Yaskawa INFORM job: B-8-08279-80-90-M.JBI

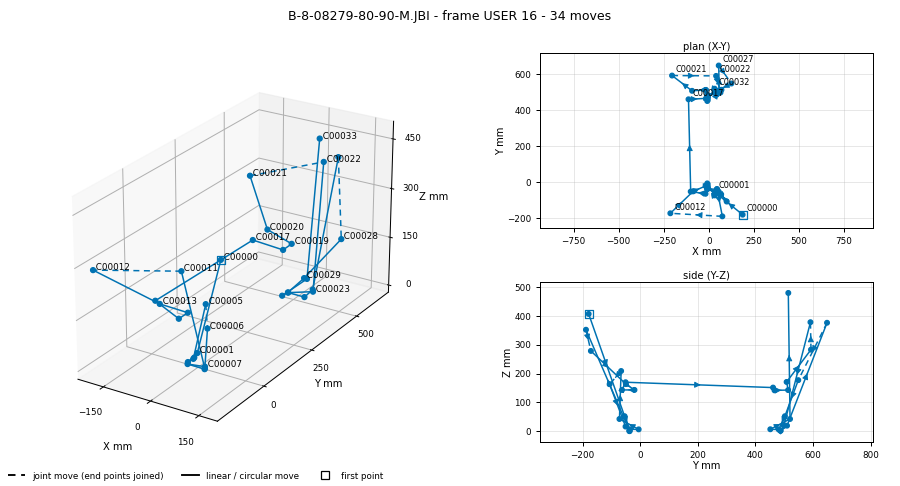
[picture p0: tool path of B-8-08279-80-90-M.JBI in frame USER 16, 34 of 34 moves have a stored position in this frame; points joined in program order, loops and branches not executed]
/JOB
//NAME B-8-08279-80-90-M
///FOLDERNAME PART_420-08279-80
//POS
///NPOS 34,0,34,0,0,0
///USER 16
///TOOL 4
///POSTYPE USER
///RECTAN
///RCONF 1,0,0,0,0,0,0,0,0,0,0,0,0,0,0,0,0,0,0,0,0,0,0,0
C00000=187.746,-179.018,407.228,-165.0003,45.0004,-0.0020
C00001=33.224,-54.308,52.156,-165.0000,45.0000,0.0000
C00002=-8.627,-36.453,6.455,-179.3917,57.1236,-36.5642
C00003=-8.579,-5.401,6.463,-179.4738,57.0912,-39.8725
C00004=32.283,-72.150,42.455,-165.0000,45.0000,0.0000
C00005=68.685,-66.272,209.042,-165.0000,45.0000,0.0000
C00006=99.538,-106.298,163.160,-166.3780,45.3490,-50.4350
C00007=54.868,-50.966,16.241,133.5610,7.6410,-152.0390
C00008=-9.081,-37.305,0.844,126.3818,11.5234,-151.1127
C00009=44.780,-37.124,0.073,126.4040,11.5044,-151.1169
C00010=45.512,-37.136,1.975,126.4030,11.5049,-151.1151
C00011=75.120,-188.373,352.355,175.5546,51.6267,-23.6686
C00012=-213.482,-171.326,278.744,154.4200,34.7310,45.4810
C00013=-87.212,-49.799,163.694,107.6090,9.3560,77.2190
C00014=-18.100,-19.955,143.362,104.0898,8.5656,76.6645
C00015=-18.153,-63.177,143.317,104.0907,8.5651,76.6651
C00016=-100.598,-50.810,170.079,107.6090,9.3560,77.2190
C00017=-112.794,461.129,151.518,107.5190,-7.4490,103.3910
C00018=-15.652,466.321,141.837,97.5692,-4.9506,104.4470
C00019=-15.525,513.463,142.905,97.5693,-4.9511,104.4481
C00020=-92.930,508.215,171.083,107.5190,-7.4490,103.3910
C00021=-203.967,592.873,283.205,107.5190,-7.4490,103.3910
C00022=40.454,590.981,378.479,-169.5230,46.0050,83.6620
C00023=64.926,498.805,18.936,-133.5620,7.6410,152.0390
C00024=-9.742,487.137,1.976,-127.4879,10.8527,151.2414
C00025=43.903,487.064,1.330,-127.4894,10.8533,151.2422
C00026=57.653,509.668,19.257,-133.5618,7.6414,152.0397
C00027=54.868,648.552,376.545,-169.5230,46.0050,83.6620
C00028=125.357,548.743,177.335,165.0000,45.0000,0.0000
C00029=33.224,502.241,52.156,165.0000,45.0000,0.0000
C00030=-7.002,480.856,5.907,165.0476,50.9832,6.6545
C00031=-8.581,451.633,6.779,162.6596,51.5731,19.7580
C00032=32.283,520.083,42.455,165.0000,45.0000,0.0000
C00033=70.181,514.089,480.075,165.0008,44.9999,-0.0009
///TOOL 0
///POSTYPE ANGLE
///ANGLE
EC00000=90.0000
///TOOL 4
EC00001=90.0000
///TOOL 0
EC00002=90.0000
EC00003=90.0000
///TOOL 4
EC00004=90.0000
EC00005=90.0000
EC00006=105.0000
EC00007=105.0000
///TOOL 0
EC00008=105.0000
EC00009=105.0000
EC00010=105.0000
EC00011=105.0000
///TOOL 4
EC00012=135.0000
EC00013=135.0000
///TOOL 0
EC00014=135.0000
EC00015=135.0000
///TOOL 4
EC00016=135.0000
EC00017=135.0000
///TOOL 0
EC00018=135.0000
EC00019=135.0000
///TOOL 4
EC00020=135.0000
EC00021=135.0000
EC00022=105.0000
EC00023=105.0000
///TOOL 0
EC00024=105.0000
EC00025=105.0000
EC00026=105.0000
///TOOL 4
EC00027=105.0000
EC00028=90.0000
EC00029=90.0000
///TOOL 0
EC00030=90.0000
EC00031=90.0000
///TOOL 4
EC00032=90.0000
///TOOL 0
EC00033=90.0000
//INST
///DATE 2021/10/29 11:36
///ATTR SC,RW,RJ
////FRAME USER 16
///GROUP1 RB1
///GROUP2 ST3
NOP
INC I005
'Path Start: PP1_1
MOVJ C00000 VJ=100.00  +MOVJ EC00000
SMOVL C00001 V=1250.0  +MOVJ EC00001
SMOVL C00002 V=1250.0  +MOVJ EC00002
ARCON ASF#(951)
SMOVL C00003 V=8.5  +MOVJ EC00003
ARCOF AEF#(951)
SMOVL C00004 V=1250.0  +MOVJ EC00004
SMOVL C00005 V=1250.0  +MOVJ EC00005
'Path End
'Path Start: PP48
MOVJ C00006 VJ=100.00  +MOVJ EC00006
SMOVL C00007 V=1250.0  +MOVJ EC00007
SMOVL C00008 V=300.0  +MOVJ EC00008
ARCON ASF#(953)
SMOVL C00009 V=15.7  +MOVJ EC00009
ARCOF AEF#(953)
SMOVL C00010 V=1250.0  +MOVJ EC00010
SMOVL C00011 V=1250.0  +MOVJ EC00011
'Path End
'Path Start: PP47
MOVJ C00012 VJ=100.00  +MOVJ EC00012
SMOVL C00013 V=1250.0  +MOVJ EC00013
SMOVL C00014 V=300.0  +MOVJ EC00014
ARCON ASF#(953)
SMOVL C00015 V=12.7  +MOVJ EC00015
ARCOF AEF#(953)
SMOVL C00016 V=1250.0  +MOVJ EC00016
'Path End
'Path Start: PP42
SMOVL C00017 V=1250.0  +MOVJ EC00017
SMOVL C00018 V=300.0  +MOVJ EC00018
ARCON ASF#(953)
SMOVL C00019 V=12.7  +MOVJ EC00019
ARCOF AEF#(953)
SMOVL C00020 V=1250.0  +MOVJ EC00020
SMOVL C00021 V=1250.0  +MOVJ EC00021
'Path End
'Path Start: PP41
MOVJ C00022 VJ=100.00  +MOVJ EC00022
SMOVL C00023 V=1250.0  +MOVJ EC00023
SMOVL C00024 V=300.0  +MOVJ EC00024
ARCON ASF#(953)
SMOVL C00025 V=15.7  +MOVJ EC00025
ARCOF AEF#(953)
SMOVL C00026 V=1250.0  +MOVJ EC00026
SMOVL C00027 V=1250.0  +MOVJ EC00027
'Path End
'Path Start: PP1
MOVJ C00028 VJ=100.00  +MOVJ EC00028
SMOVL C00029 V=1250.0  +MOVJ EC00029
SMOVL C00030 V=1250.0  +MOVJ EC00030
ARCON ASF#(951)
SMOVL C00031 V=8.5  +MOVJ EC00031
ARCOF AEF#(951)
SMOVL C00032 V=1250.0  +MOVJ EC00032
SMOVL C00033 V=1250.0  +MOVJ EC00033
'Path End
END
